FUNCTION_BLOCK FB_GridPointFIFO
VAR_OUTPUT
	nCount    : UINT;                 // Fill level
END_VAR
VAR
	sBuffer 	: ARRAY[0..(MAX_BUFFER_SIZE-1)] OF ST_GridPoint;
	nHeadPtr  : UINT := 0;            // Point to the first non-empty idx
	nTailPtr  : UINT := 0;            // Pointer to the first free idx
  _bError   : BOOL;
END_VAR
VAR CONSTANT
	MAX_BUFFER_SIZE   : UINT := 500;  // max. buffer size
END_VAR

PROPERTY bError : BOOL
GET
bError := _bError;
END_GET
END_PROPERTY

(*
  Get point from fifo queue. 
  :return: TRUE on success
*)
METHOD Pop : BOOL
VAR_OUTPUT
	sGridPoint : ST_GridPoint;
END_VAR
IF nCount = 0 THEN
  F_LogError('FB_DeformationPointFIFO is empty, cannot return an element');
  _bError := TRUE; 
  RETURN;
END_IF

sGridPoint := sBuffer[nTailPtr];
nTailPtr := (nTailPtr + 1) MOD MAX_BUFFER_SIZE;
nCount := nCount - 1;
_bError := FALSE;
Pop := TRUE;
END_METHOD

(*
  Add a new point to the fifo queue.
  :return: TRUE on success.
*)
METHOD Push : BOOL
VAR_INPUT
	sNewPoint : ST_GridPoint;
END_VAR
IF nCount >= MAX_BUFFER_SIZE THEN
  F_LogError('FB_DeformationPointFIFO overflow, element ignored');
  _bError := TRUE;
  RETURN;
END_IF

sBuffer[nHeadPtr] := sNewPoint;
nHeadPtr := (nHeadPtr + 1) MOD MAX_BUFFER_SIZE;
nCount := nCount + 1;
_bError := FALSE;
Push := TRUE;
END_METHOD

METHOD Reset : BOOL
VAR_INPUT
END_VAR
nTailPtr := 0;
nHeadPtr := 0;
nCount := 0;
_bError := 0;
END_METHOD

END_FUNCTION_BLOCK

(* stored: Version 1.1.0.1, ProductVersion 3.1.4024.3
   POU FB_GridPointFIFO: Id {8c086e8c-cff0-4648-8bd3-98b05260a0a4}, SpecialFunc None
   Property bError: Id {a012fb6e-0800-42f3-8d79-34f01a1bdc2c}
   Get Get: Id {c375fde1-e151-42cf-bd1e-70a77c9ac55a}
   Method Pop: Id {a098839a-72ec-4ab0-b04f-472da796b700}
   Method Push: Id {91a35e6a-70a9-47bd-a034-e22fe4faa50f}
   Method Reset: Id {9fb5f1a7-e929-4852-9362-6fab0cbb7438} *)
